{attribute 'qualified_only'}
VAR_GLOBAL
	// Konfiguration
	stConfig: ST_Config := (rLaenge := 300, rBreite := 200, rDicke := 30);
END_VAR

(* stored: Version 1.1.0.1, ProductVersion 3.1.4024.3
   GVL GVL_Config: Id {df27e69c-833e-4f2b-b7a2-5ebc50e8e97a} *)
